{attribute addProperty BoxType "EL3773-0000-0016"}
{attribute addProperty Id "U3_STATUSAT %I*U3_STATUS_F9B4A013162"}
{attribute addProperty CRC "4249091381"}
{attribute addProperty SizeInBites "16"}
{attribute addProperty SizeInBytes "2"}
TYPE L3_Voltage_Status_FD43FD35 :
STRUCT
	{attribute addProperty Name "U3_STATUS"}
	U3_STATUS AT %I* : U3_STATUS_F9B4A013;
END_STRUCT
END_TYPE

(* stored: Version 1.2.0.0, ProductVersion 3.1.4024.9
   DUT L3_Voltage_Status_FD43FD35: Id {209539fe-b6ba-47e7-a4d5-486dc0b49fbe} *)
